TYPE csp_case_feed_connection_status_enum :
(		
	CSP_CASE_FEED_STATUS_CONNECTION_START							:= 0,
	CSP_CASE_FEED_STATUS_CONNECTION_ENGAGE							:= 10,
	CSP_CASE_FEED_STATUS_CONNECTION_ENGAGED							:= 20,
	CSP_CASE_FEED_STATUS_CONNECTION_CHECK_CHANGE_CAM				:= 30,
	CSP_CASE_FEED_STATUS_CONNECTION_CHANGE_CAM						:= 40,
	CSP_CASE_FEED_STATUS_CONNECTION_WAIT_NEW_CAM					:= 50,
	CSP_CASE_FEED_STATUS_CONNECTION_STOPPING						:= 100,
	CSP_CASE_FEED_STATUS_CONNECTION_STOPPED							:= 110,
	CSP_CASE_FEED_STATUS_CONNECTION_REJECT_STEP1					:= 201,
	CSP_CASE_FEED_STATUS_CONNECTION_REJECT_STEP2					:= 202,
	CSP_CASE_FEED_STATUS_CONNECTION_REJECT_STEP3					:= 203,
	CSP_CASE_FEED_STATUS_CONNECTION_REJECT_STEP4					:= 204,
	CSP_CASE_FEED_STATUS_CONNECTION_REJECT_STEP5					:= 205,
	CSP_CASE_FEED_STATUS_CONNECTION_REJECT_STEP6					:= 206,
	CSP_CASE_FEED_STATUS_CONNECTION_REJECT_STEP7					:= 207,
	CSP_CASE_FEED_STATUS_CONNECTION_REJECT_STEP8					:= 208,
	CSP_CASE_FEED_STATUS_CONNECTION_REJECT_STEP9					:= 209,	
	CSP_CASE_FEED_STATUS_CONNECTION_DONE 							:= 900,
	CSP_CASE_FEED_STATUS_CONNECTION_ERROR 							:= 999
) := CSP_CASE_FEED_STATUS_CONNECTION_START;
END_TYPE

(* stored: Version 1.1.0.1, ProductVersion 3.1.4022.12
   DUT csp_case_feed_connection_status_enum: Id {ff0d9565-bd4b-4b29-8cff-385bd311d97d} *)
